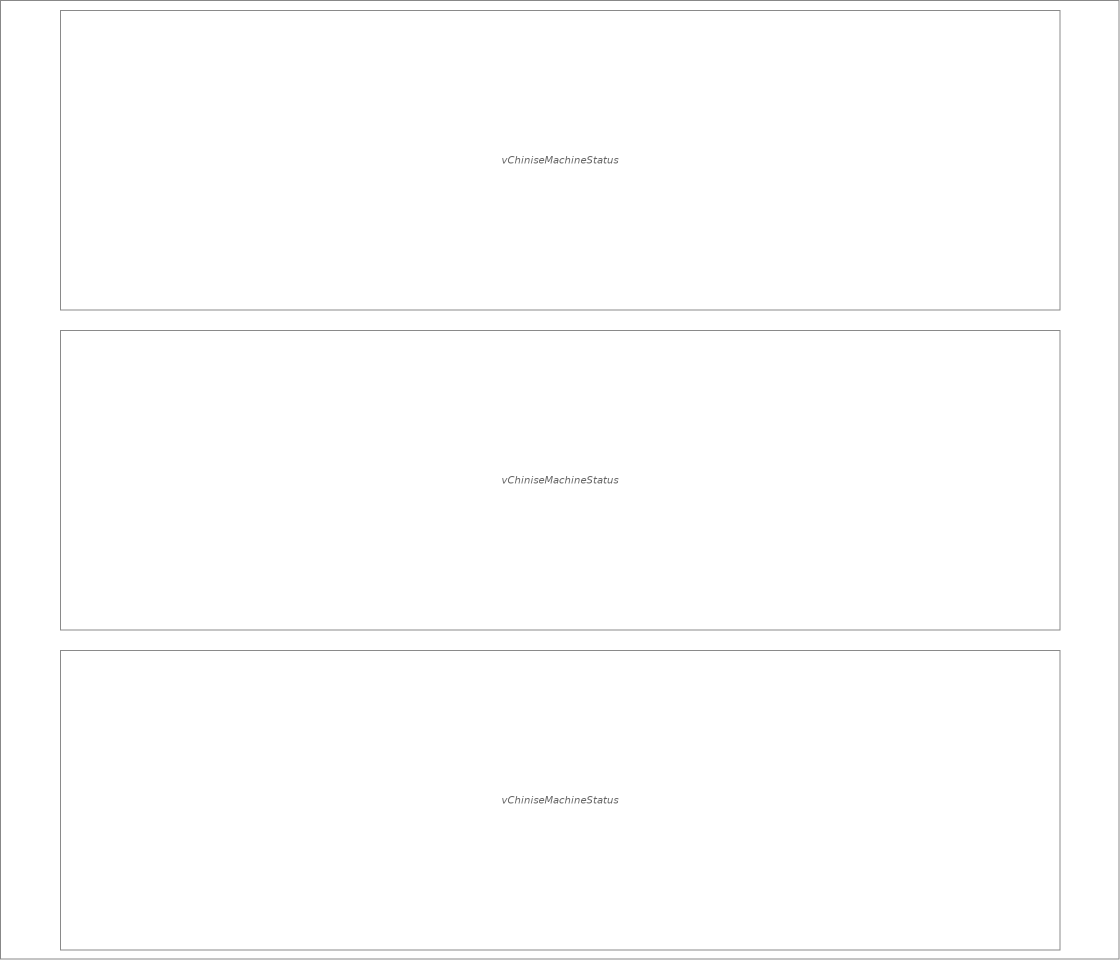
VISUALIZATION vFrameFillingLine_1  // 1120x960
VAR_IN_OUT

END_VAR
VAR
	iFiller_A 	: UINT := 0;
	iCork 		: UINT := 1;
	iFiller_B 	: UINT := 2;
	iSticker	: UINT := 3;
	iLaser		: UINT := 4;
END_VAR
    Frame (60,10 1000x300)
        shows vChiniseMachineStatus(stData := GVL.st_Filler_A_MachineSettings.stPimData, fbPIM := MAIN.fb_Filler_A_Station, iActualMachine := iFiller_A, fbModbusTCP := MAIN.fb_Filler_A_Machine.fbModbuCommunication, bTurnOnCommunication := GVL.st_Filler_A_MachineSettings.bCommunicationActive, iCommunicationCycleTime := GVL.st_Filler_A_MachineSettings.iCommunicationCycleTime)
    Frame (60,330 1000x300)
        shows vChiniseMachineStatus(stData := GVL.st_Cork_MachineSettings.stPimData, fbPIM := MAIN.fb_Cork_Station, iActualMachine := iCork, fbModbusTCP := MAIN.fb_Cork_Machine.fbModbuCommunication, bTurnOnCommunication := GVL.st_Cork_MachineSettings.bCommunicationActive, iCommunicationCycleTime := GVL.st_Cork_MachineSettings.iCommunicationCycleTime)
    Frame (60,650 1000x300)
        shows vChiniseMachineStatus(stData := GVL.st_Filler_B_MachineSettings.stPimData, fbPIM := MAIN.fb_Filler_B_Station, iActualMachine := iFiller_B, fbModbusTCP := MAIN.fb_Filler_B_Machine.fbModbuCommunication, bTurnOnCommunication := GVL.st_Filler_B_MachineSettings.bCommunicationActive, iCommunicationCycleTime := GVL.st_Filler_B_MachineSettings.iCommunicationCycleTime)
END_VISUALIZATION

(* stored: Version 1.1.0.1, ProductVersion 3.1.4024.13
   Visu vFrameFillingLine_1: Id {6907ec24-c443-4c27-9dc5-7ee0f0306b7e} *)
